SUBAPPLICATION Uebung_128 (* Übung zu ISOBUS Send Message GLOBAL *)
  (* Standard: 61499-2; Description: Copyright (c) 2025 Meisterschulen am Ostbahnhof This program and the accompanying materials are made available under the terms of the Eclipse Public License 2.0 which is available at https://www.eclipse.org/legal/epl-2.0/ SPDX-License-Identifier: EPL-2.0 *)
  (* Version 1.0, 2023-10-23, Franz Höpfinger, Meisterschulen am Ostbahnhof *)
  IMPORT isobus::pgn::ADDRESS::GLOBAL_A;
  IMPORT isobus::pgn::ISOUSERHOME_e::thisMember;
  IMPORT isobus::pgn::ISO_CAN_NODE::NODE1;
  IMPORT logiBUS::io::DI::logiBUS_DI::Input_I1;
  IMPORT logiBUS::io::DI::logiBUS_DI_Events::BUTTON_SINGLE_CLICK;
  IMPORT uebungen::Filter::FLT_ALL_PASS;
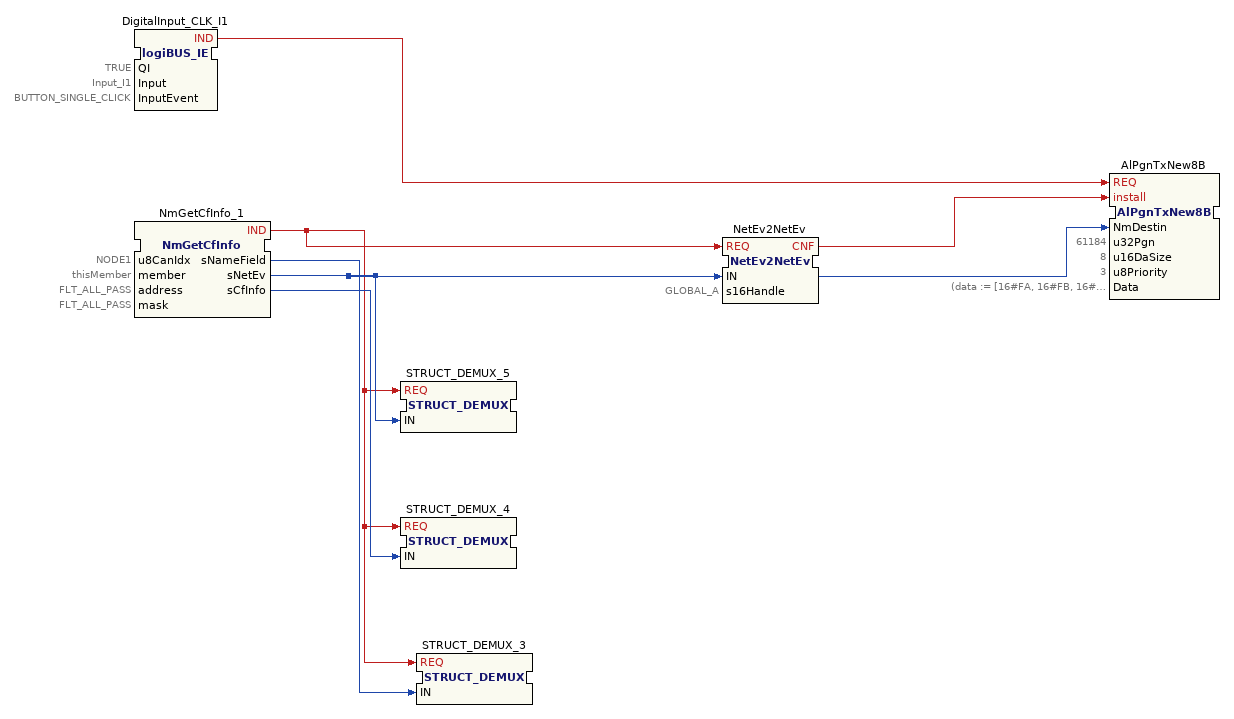
  FBS
    STRUCT_DEMUX_3 : eclipse4diac::convert::STRUCT_DEMUX; {SET_ATTRIBUTE(StructuredType, isobus::pgn::NAMEFIELD_T)}
    NmGetCfInfo_1 : isobus::pgn::NmGetCfInfo(u8CanIdx := NODE1, member := thisMember, address := FLT_ALL_PASS, mask := FLT_ALL_PASS);
    STRUCT_DEMUX_4 : eclipse4diac::convert::STRUCT_DEMUX; {SET_ATTRIBUTE(StructuredType, isobus::pgn::CF_INFO_T)}
    STRUCT_DEMUX_5 : eclipse4diac::convert::STRUCT_DEMUX; {SET_ATTRIBUTE(StructuredType, isobus::pgn::ISONETEVENT_T)}
    AlPgnTxNew8B : isobus::pgn::tx::AlPgnTxNew8B(u32Pgn := 61184, u16DaSize := 8, u8Priority := 3, Data := (data := [16#FA, 16#FB, 16#FC, 16#FD, 16#FE, 16#FF, 16#F1, 16#F2]));
    DigitalInput_CLK_I1 : logiBUS::io::DI::logiBUS_IE(QI := TRUE, Input := Input_I1, InputEvent := BUTTON_SINGLE_CLICK);
    NetEv2NetEv : isobus::PGN::NetEv2NetEv(s16Handle := GLOBAL_A);
  END_FBS
  EVENT_CONNECTIONS
    NmGetCfInfo_1.IND TO STRUCT_DEMUX_3.REQ;
    NmGetCfInfo_1.IND TO STRUCT_DEMUX_4.REQ;
    NmGetCfInfo_1.IND TO STRUCT_DEMUX_5.REQ;
    NmGetCfInfo_1.IND TO NetEv2NetEv.REQ;
    DigitalInput_CLK_I1.IND TO AlPgnTxNew8B.REQ;
    NetEv2NetEv.CNF TO AlPgnTxNew8B.install;
  END_CONNECTIONS
  DATA_CONNECTIONS
    NmGetCfInfo_1.sNameField TO STRUCT_DEMUX_3.IN;
    NmGetCfInfo_1.sNetEv TO STRUCT_DEMUX_5.IN;
    NmGetCfInfo_1.sCfInfo TO STRUCT_DEMUX_4.IN;
    NmGetCfInfo_1.sNetEv TO NetEv2NetEv.IN;
    NetEv2NetEv. TO AlPgnTxNew8B.NmDestin;
  END_CONNECTIONS
END_SUBAPPLICATION
